SUBAPPLICATION Uebung_011b1_PHYS (* Numeric Value Input ADD (PHYS) *)
  (* Standard: 61499-2; Description: Copyright (c) 2026 Meisterschulen am Ostbahnhof This program and the accompanying materials are made available under the terms of the Eclipse Public License 2.0 which is available at https://www.eclipse.org/legal/epl-2.0/ SPDX-License-Identifier: EPL-2.0 *)
  (* Version 1.0, 2026-04-24, Franz Höpfinger, Meisterschulen am Ostbahnhof, PHYS variant of Uebung_011b1 with REAL arithmetic *)
  PACKAGE Uebungen;
  IMPORT Uebungen::const::UT::DefaultPool_Numeric::InputNumber_I3_N;
  IMPORT Uebungen::const::UT::DefaultPool_Numeric::InputNumber_I4_N;
  IMPORT Uebungen::const::UT::DefaultPool_Numeric::OutputNumber_N3_N;
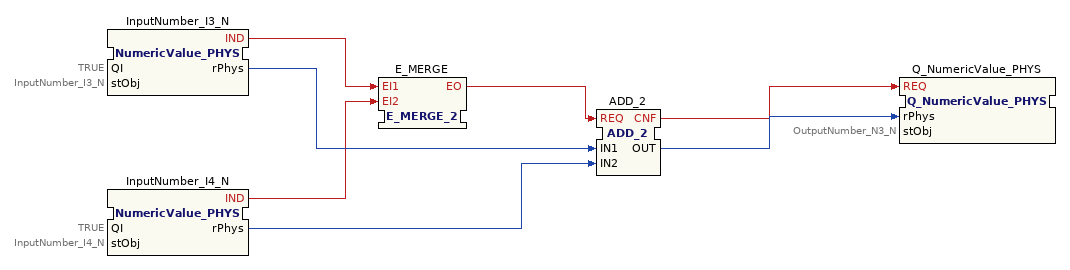
  FBS
    InputNumber_I3_N : isobus::UT::io::NumericValue::NumericValue_PHYS(QI := TRUE, stObj := InputNumber_I3_N);
    InputNumber_I4_N : isobus::UT::io::NumericValue::NumericValue_PHYS(QI := TRUE, stObj := InputNumber_I4_N);
    ADD_2 : iec61131::arithmetic::ADD_2;
    Q_NumericValue_PHYS : isobus::UT::Q::Q_NumericValue_PHYS(stObj := OutputNumber_N3_N);
    E_MERGE : iec61499::events::E_MERGE_2;
  END_FBS
  EVENT_CONNECTIONS
    ADD_2.CNF TO Q_NumericValue_PHYS.REQ;
    E_MERGE.EO TO ADD_2.REQ;
    InputNumber_I3_N.IND TO E_MERGE.EI1;
    InputNumber_I4_N.IND TO E_MERGE.EI2;
  END_CONNECTIONS
  DATA_CONNECTIONS
    InputNumber_I3_N.rPhys TO ADD_2.IN1;
    ADD_2.OUT TO Q_NumericValue_PHYS.rPhys;
    InputNumber_I4_N.rPhys TO ADD_2.IN2;
  END_CONNECTIONS
END_SUBAPPLICATION
